Fanuc KAREL source: ko00071.KL

-- PROVISIONAL review KL for V1013-1; original PC SHA256 11671012799944a786f9506cbfb360230daba53e8d4b4bf126e09e64d13e1e88
-- Incomplete behavior may be omitted. Consult companion uncertainty JSON. Do not deploy.
PROGRAM KO00071
%NOLOCKGROUP
BEGIN
  -- UNRESOLVED_PC offsets 5-12; opcodes 9D,23
  -- UNRESOLVED_PC offsets 17-66; opcodes 27,22,1C,27,49,7E,AD,22,31,7E,4A
  -- UNRESOLVED_PC offsets 71-75; opcodes 7F
END KO00071
